FUNCTION F_CheckIndexBounds : INT
VAR_INPUT
	lowerbound		: 	INT;
	upperbound		:   INT;
END_VAR
VAR_IN_OUT
	index			: 	INT;
END_VAR

IF  index < lowerbound THEN
	F_CheckIndexBounds := lowerbound;
	index 		:= lowerbound;
ELSIF  index > upperbound THEN
	F_CheckIndexBounds := upperbound;
	index 		:= upperbound;
ELSE  
	F_CheckIndexBounds := index;
END_IF

END_FUNCTION

(* stored: Version 1.1.0.1, ProductVersion 3.1.4022.6
   POU F_CheckIndexBounds: Id {d76e7c2f-cc9d-42a4-a3cb-492ecfa98d49}, SpecialFunc None *)
